RoboDK station: Welding Operation.rdk

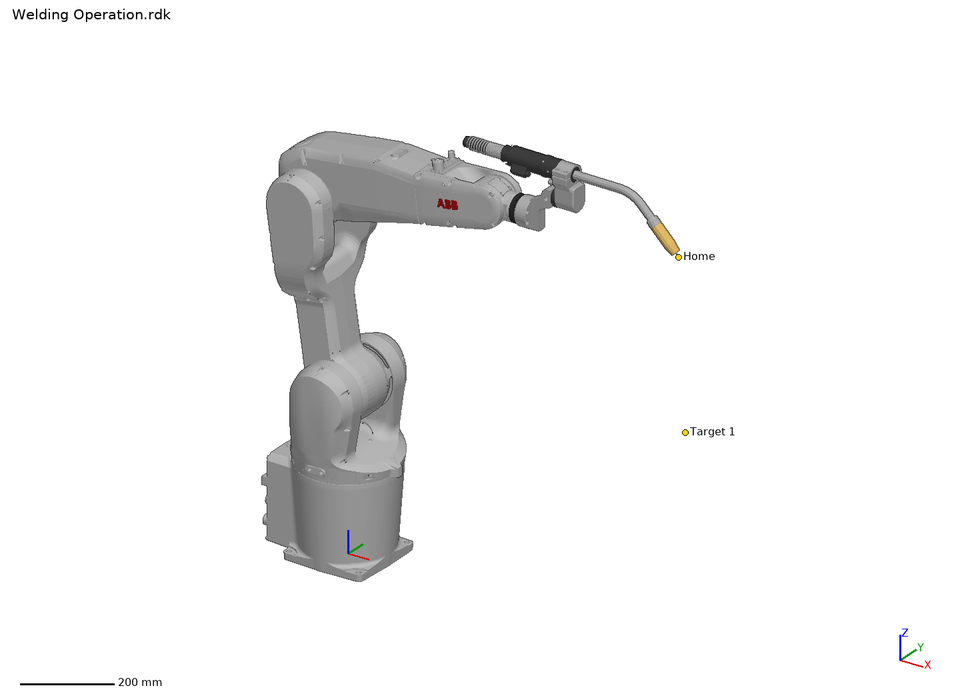
[picture v0: the station drawn from its stored meshes, robots at their saved joint values, targets as dots, program paths as lines]
Station Demo Program new robot (saved by RoboDK 5.2.1). Poses are relative to the parent item; angles as X-Y-Z fixed-axis rotations.
Station parameters (name, value as stored): LIN64
  - frame ABB IRB 1200-5/0.9 Base at (0, 0, 0) mm
    - robot ABB IRB 1200-5/0.9: 6 axes, payload 5 kg, reach 901 mm, repeatability 0.02 mm, weight 52 kg
        modified DH rows (alpha deg, a mm, theta deg, d mm): 0, 0, 0, 399; -90, 0, -90, 0; 0, 448, 0, 0; -90, 42, 0, 451; 90, 0, 0, 0; -90, 0, 180, 82
        joint limits [-170, -100, -200, -270, -130, -360] to [170, 130, 70, 270, 130, 360]; home [0, 0, 0, 0, 0, 0]; saved at [0, -8.567, 1.423, 0, 7.143, 0]
      - tool Weld Torch Abicor Binzel 45deg, TCP at (0, 0, 400) mm, rotated rx 0 ry 45 rz 0 deg, size 179.1 x 69.8 x 552.4 mm
    - target Home (Cartesian target) at (857.54, 0, 939.76) mm, rotated rx -180 ry 45 rz -180 deg; joints [0, -5.068, -1.138, 0, 6.206, 0] of ABB IRB 1200-5/0.9
    - target Target 1 (Cartesian target) at (878.55, -5.8, 533.14) mm, rotated rx 180 ry 45 rz 180 deg; joints [-0.839, 8.401, 39.944, -1.122, -48.35, 0.746] of ABB IRB 1200-5/0.9
  - Python program Weld Progam Code (listed below)

--- Python program Weld Progam Code ---
# Type help("robolink") or help("robodk") for more information
# Press F5 to run the script
# Documentation: https://robodk.com/doc/en/RoboDK-API.html
# Reference:     https://robodk.com/doc/en/PythonAPI/index.html
# Note: It is not required to keep a copy of this file, your python script is saved with the station
from robolink import *    # RoboDK API
from robodk import *      # Robot toolbox

# The Robolink() module is what is used to interact and communicate with RoboDK
RDK = Robolink()

# Assigning the robot item to a variable
robot = RDK.Item('ABB IRB 1200-5/0.9')

# Using the Robolink module we can get the Home target and the welding target(s)
# from RoboDK and assign them both to a variable
home = RDK.Item('Home')
target = RDK.Item('Target 1')

# Using the Robolink module we are able to get the position of the target in space
# from the RoboDK simulation environment
# in the form of a 4x4 matrix and then we save this to a variable
reference_pose = target.Pose()

# Using the Robolink module we first move the robot arm to the 'Home' position
# and then to the 'Target 1' position
robot.MoveJ(home)
robot.MoveJ(target)

# From the RoboDK module we're able to use a message box
# to collect the desired amount of vertices the shape should have from the user
# This can be used to make different shapes including a circle, triangle, square etc.
num_vertices = mbox("Enter then number of vertices", entry=True)
num_vertices = int(num_vertices)

# Using both the RoboDK and the Robolink  module we're able to
# make a hexagon shape around the center of the selected target
for i in range(num_vertices+1):
    ang = i*2*pi/num_vertices      # used to obtain angles: 0, 60, 120, ..., 360
    vertex_pose = reference_pose*rotz(ang)*transl(300, 0, 0)*rotz(-ang)
    robot.MoveL(vertex_pose)

# Finally we move the robot arm back to the target position and then to the home
# position and the program ends.
robot.MoveL(target)
robot.MoveJ(home)
